{attribute 'qualified_only'}
{attribute 'strict'}
TYPE
    eCUMode :
    (
        NoMode         := 0,
        GroundMode     := 10,
        GroundModeDone := 15,
        AutomatMode    := 20,
        ManualMode     := 30
    );
END_TYPE

(* stored: Version 1.1.0.1
   DUT eCUMode: Id {95533cd7-3a00-4614-8cf9-ed41b8c0fc55} *)
